// Mitsubishi GX Works2 project: 250626_Robot+Cylinders   PLC: Q02U

PROGRAM MAIN
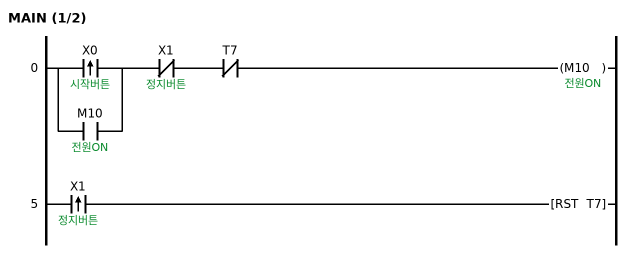
0     LDP     X0  ; 시작버튼
      OR      M10  ; 전원ON
      ANI     X1  ; 정지버튼
      ANI     T7
      OUT     M10  ; 전원ON
5     LDP     X1  ; 정지버튼
      RST     T7
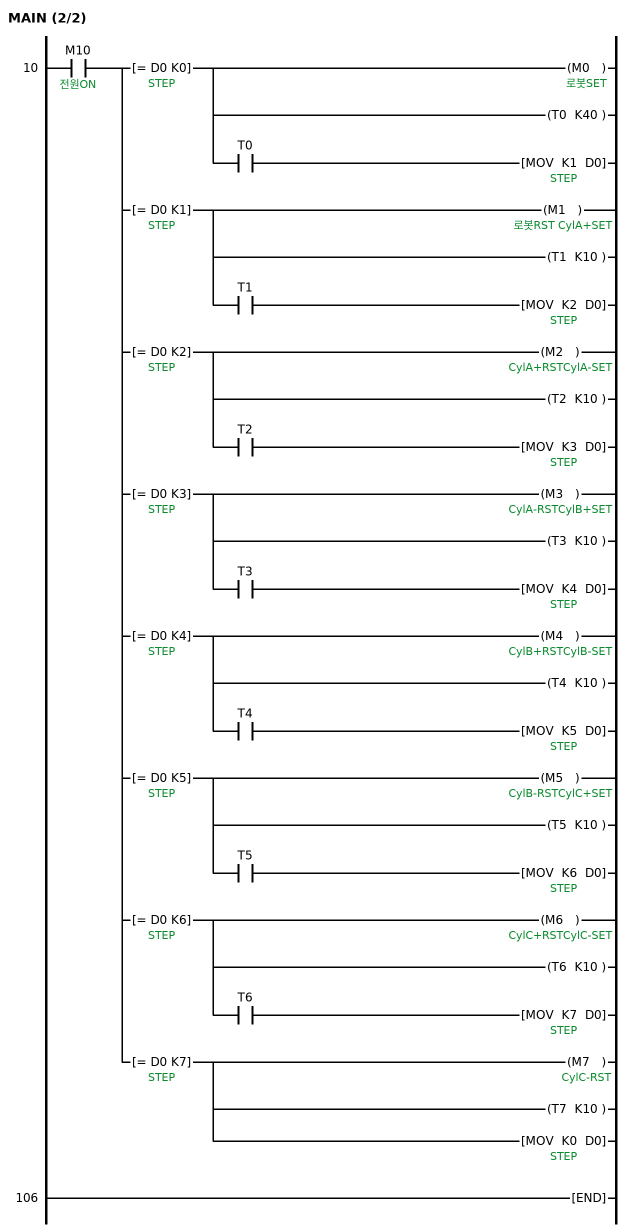
10    LD      M10  ; 전원ON
      MPS
      AND=    D0 K0  ; STEP
      OUT     M0  ; 로봇SET
      OUT     T0 K40
      AND     T0
      MOV     K1 D0
      MRD
      AND=    D0 K1  ; STEP
      OUT     M1  ; 로봇RST CylA+SET
      OUT     T1 K10
      AND     T1
      MOV     K2 D0
      MRD
      AND=    D0 K2  ; STEP
      OUT     M2  ; CylA+RSTCylA-SET
      OUT     T2 K10
      AND     T2
      MOV     K3 D0
      MRD
      AND=    D0 K3  ; STEP
      OUT     M3  ; CylA-RSTCylB+SET
      OUT     T3 K10
      AND     T3
      MOV     K4 D0
      MRD
      AND=    D0 K4  ; STEP
      OUT     M4  ; CylB+RSTCylB-SET
      OUT     T4 K10
      AND     T4
      MOV     K5 D0
      MRD
      AND=    D0 K5  ; STEP
      OUT     M5  ; CylB-RSTCylC+SET
      OUT     T5 K10
      AND     T5
      MOV     K6 D0
      MRD
      AND=    D0 K6  ; STEP
      OUT     M6  ; CylC+RSTCylC-SET
      OUT     T6 K10
      AND     T6
      MOV     K7 D0
      MPP
      AND=    D0 K7  ; STEP
      OUT     M7  ; CylC-RST
      OUT     T7 K10
      MOV     K0 D0
106   END
END_PROGRAM

PROGRAM MAIN1
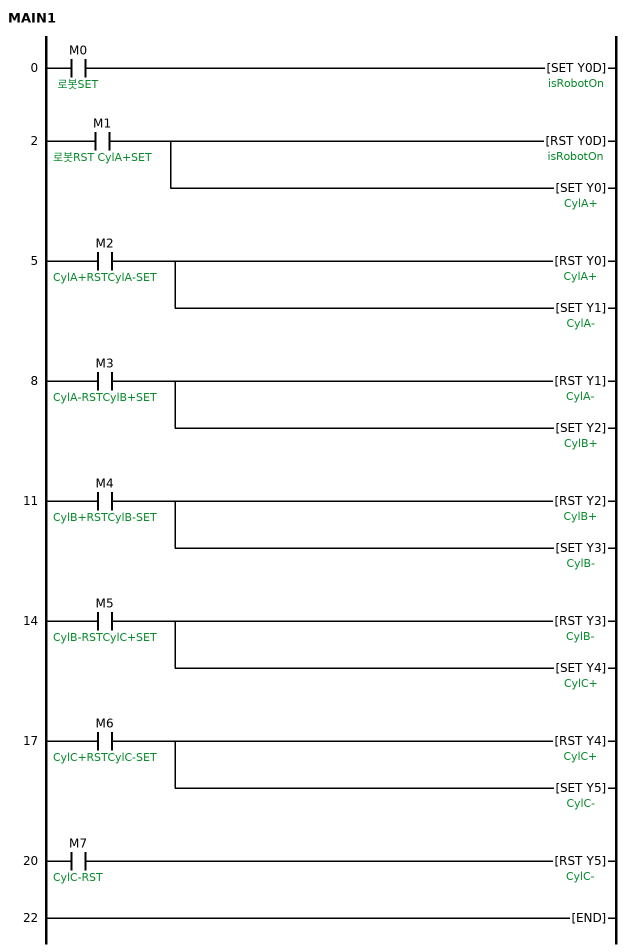
0     LD      M0  ; 로봇SET
      SET     Y0D  ; isRobotOn
2     LD      M1  ; 로봇RST CylA+SET
      RST     Y0D  ; isRobotOn
      SET     Y0  ; CylA+
5     LD      M2  ; CylA+RSTCylA-SET
      RST     Y0  ; CylA+
      SET     Y1  ; CylA-
8     LD      M3  ; CylA-RSTCylB+SET
      RST     Y1  ; CylA-
      SET     Y2  ; CylB+
11    LD      M4  ; CylB+RSTCylB-SET
      RST     Y2  ; CylB+
      SET     Y3  ; CylB-
14    LD      M5  ; CylB-RSTCylC+SET
      RST     Y3  ; CylB-
      SET     Y4  ; CylC+
17    LD      M6  ; CylC+RSTCylC-SET
      RST     Y4  ; CylC+
      SET     Y5  ; CylC-
20    LD      M7  ; CylC-RST
      RST     Y5  ; CylC-
22    END
END_PROGRAM

// device comments not shown above
X2  ; 긴급정지버튼
X19  ; 근접센서ON
X1A  ; 금속센서ON
Y6  ; CylD+
Y7  ; CylD-
Y8  ; isCW
Y9  ; isCCW
Y0A  ; isRedLampOn
Y0B  ; isYellowLampOn
Y0C  ; isGreenLampOn
